FUNCTION_BLOCK IAS_Skill_DEMUX (* Composite Function Block Type *)
  (* Standard: 61499-2 *)
  (* Version 1.0, 2019-07-03, dorofeev *)
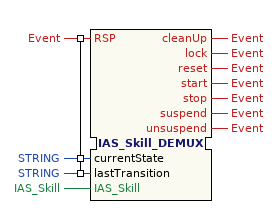
  EVENT_INPUT
    RSP WITH currentState, lastTransition;
  END_EVENT
  EVENT_OUTPUT
    cleanUp; (* Initialization Confirm *)
    lock;
    reset;
    start;
    stop;
    suspend;
    unsuspend;
  END_EVENT
  VAR_INPUT
    currentState : STRING;
    lastTransition : STRING;
  END_VAR
  SOCKETS
    IAS_Skill : IAS_Skill;
  END_SOCKETS
  EVENT_CONNECTIONS
    IAS_Skill.cleanUp TO cleanUp;
    IAS_Skill.lock TO lock;
    IAS_Skill.reset TO reset;
    IAS_Skill.start TO start;
    IAS_Skill.stop TO stop;
    IAS_Skill.suspend TO suspend;
    IAS_Skill.unsuspend TO unsuspend;
    RSP TO IAS_Skill.RSP;
  END_CONNECTIONS
  DATA_CONNECTIONS
    currentState TO IAS_Skill.currentState;
    lastTransition TO IAS_Skill.lastTransition;
  END_CONNECTIONS
END_FUNCTION_BLOCK
